FUNCTION alg_a_Dstartled : BOOL
VAR_INPUT
	state: STATE;
END_VAR

alg_a_Dstartled := alg_M_example_controller_a_Dstartled(state);

END_FUNCTION

(* stored: Version 1.1.0.1, ProductVersion 3.1.4022.18
   POU alg_a_Dstartled: Id {90248504-e61b-4862-97e1-bd1f834c9364}, SpecialFunc None *)
